Universal Robots PolyScope program: pick_repeat.urp

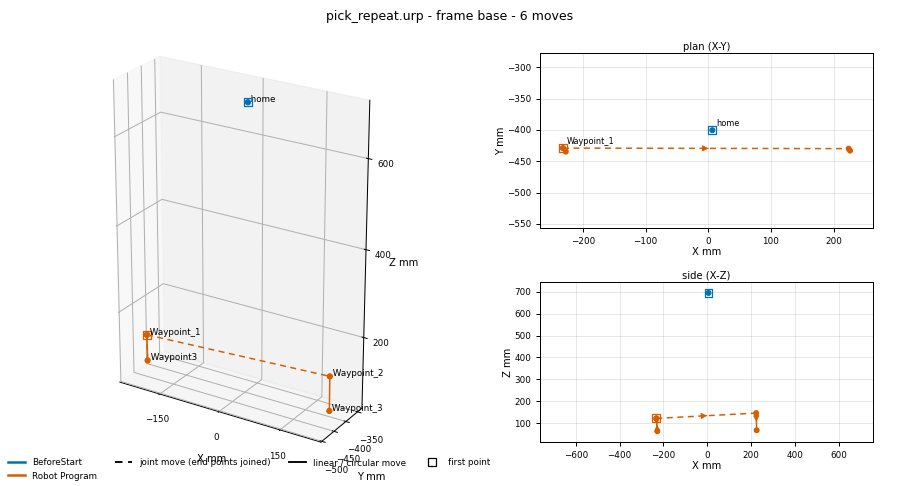
[picture p0: tool path of pick_repeat.urp in frame base, 6 of 6 moves have a stored position in this frame; points joined in program order, loops and branches not executed]
Program pick_repeat (installation=default directory=/programs createdIn=5.14.5 lastSavedIn=5.14.5 robotSerialNumber=20195300809)
Calibrated DH parameters: a=[-0.000085, -0.20076, -0.212369, 0.000121, -0.000118, 0]; d=[0.15185, -26.306375, 24.753047, 1.684739, 0.085386, 0.092088]; alpha=[1.572149, -0.00522, -0.011864, 1.571339, -1.571085, 0]; deltaTheta=[0, 0.599885, -0.513355, -0.086555, 0.000006, 0]
InitVariablesNode
BeforeStart
  MoveJ speed 60 deg/s, acceleration 80 deg/s^2 (useActiveTCP=true) feature=Base
    Waypoint home: TCP in base x=6.411 y=-400.316 z=694.751 mm, rx=-0.0179 ry=2.2101 rz=-2.2165 rad; joints [0.003, -90, 0.001, -89.999, 0, 0.002] deg; TCP offset x=0 y=0 z=177.62 mm, rx=0 ry=0 rz=0 rad
  URCap Gripper Activate (Robotiq_Grippers, Robotiq Inc.) dataModel(ResetAndActivateKey=false)
Robot Program (runOnlyOnce=false)
  URCap Gripper (Robotiq_Grippers, Robotiq Inc.) dataModel(position=0.0, force=0.0, speed=0.0, positionInDouble=0.0, forceInDouble=0.0, speedInDouble=0.0, slaveIds=[9], blocking=true)
  Set DigitalOutput pin=digital_out[0]; digitalValue=1
  Wait DigitalInput pin=digital_in[0]; digitalValue=0
  If digital_in[0]≟0
    Set DigitalOutput pin=digital_out[0]; digitalValue=0
  MoveJ speed 60 deg/s, acceleration 80 deg/s^2 (useActiveTCP=true) feature=Base
    Waypoint Waypoint_1: TCP in base x=-231.969 y=-428.883 z=121.822 mm, rx=-0.0883 ry=3.1015 rz=-0.1202 rad; joints [-104.887, -132.675, -32.103, -101.515, 92.471, -17.533] deg
  MoveL speed 250 mm/s, acceleration 1200 mm/s^2 (useActiveTCP=true) feature=Base
    Waypoint Waypoint3: TCP in base x=-227.492 y=-434.612 z=63.315 mm, rx=-0.0163 ry=3.1376 rz=0.0818 rad; joints [-102.075, -141.358, -29.172, -102.411, 88.721, -12.128] deg
  URCap Gripper (Robotiq_Grippers, Robotiq Inc.) dataModel(position=100.0, force=0.0, speed=0.0, positionInDouble=100.0, forceInDouble=0.0, speedInDouble=0.0, slaveIds=[9], blocking=true)
  MoveJ speed 60 deg/s, acceleration 80 deg/s^2 (useActiveTCP=true) feature=Base
    Waypoint Waypoint_1: TCP in base x=-231.969 y=-428.883 z=121.822 mm, rx=-0.0883 ry=3.1015 rz=-0.1202 rad; joints [-104.887, -132.675, -32.103, -101.515, 92.471, -17.533] deg
  MoveJ speed 60 deg/s, acceleration 80 deg/s^2 (useActiveTCP=true) feature=Base
    Waypoint Waypoint_2: TCP in base x=224.109 y=-429.754 z=146.092 mm, rx=2.1045 ry=2.1697 rz=-0.2208 rad; joints [103.91, -57.246, 46.868, -89.465, -94.59, 101.84] deg; TCP offset x=0 y=0 z=177.62 mm, rx=0 ry=0 rz=0 rad
  MoveL speed 250 mm/s, acceleration 1200 mm/s^2 (useActiveTCP=true) feature=Base
    Waypoint Waypoint_3: TCP in base x=226.237 y=-432.95 z=67.637 mm, rx=2.2225 ry=2.2103 rz=-0.0345 rad; joints [102.468, -46.197, 44.471, -89.3, -91.749, 102.751] deg; TCP offset x=0 y=0 z=177.62 mm, rx=0 ry=0 rz=0 rad
